FUNCTION_BLOCK TEvent_SecondsChanged EXTENDS TEventBase IMPLEMENTS IEvent
VAR
	Now: TIMESTRUCT;
    Handler : IEventHandler_OnSecondsChanged;
END_VAR

METHOD  CallHandler
VAR_INPUT
    HandlerBase : IEventHandlerBase;
END_VAR
IF __QUERYINTERFACE(HandlerBase,Handler) THEN
    Handler.OnSecondsChanged(Now);
END_IF
END_METHOD

METHOD  IsHandlerSupported : BOOL
VAR_INPUT
    EventHandler : IEventHandlerBase;
END_VAR
IF __QUERYINTERFACE(EventHandler,Handler) THEN
    IsHandlerSupported := TRUE;
END_IF
END_METHOD

METHOD RaiseEx
VAR_INPUT
	Now: TIMESTRUCT;
END_VAR
THIS^.Now := Now;
SUPER^.Raise();
END_METHOD

END_FUNCTION_BLOCK

(* stored: Version 1.1.0.1, ProductVersion 3.1.4024.3
   POU TEvent_SecondsChanged: Id {57a76d21-1795-042e-20b6-0c8a44b55557}, SpecialFunc None
   Method CallHandler: Id {78966186-ac6c-0d07-2492-7cf5120a8188}
   Method IsHandlerSupported: Id {02ca237e-cffb-0ad8-1722-70a4c95ed470}
   Method RaiseEx: Id {a20063a4-20f5-088c-0098-002c926dc4b1} *)
